PROGRAM MAIN
VAR
END_VAR

END_PROGRAM

(* stored: Version 1.1.0.1
   POU MAIN: Id {2fb17c1a-5e80-4d1a-bf35-24246e7b43b9} *)
